TYPE CamTableSelectCMD_typ :
	STRUCT
		
		Start 		: BOOL;

	END_STRUCT
END_TYPE

(* stored: Version 1.1.0.1, ProductVersion 3.1.4024.3
   DUT CamTableSelectCMD_typ: Id {6bdf3301-4a6d-0df5-139f-67daa460fb55} *)
